(* IEC 61131-3 sources: RL_MAR/experiments/comparison/llm4plc/results/gpt-4o-mini_20260506_100619/20260506_103717, 4 files *)

(* ---- generated_code_iteration_0.st ---- *)
ructured-text
START_ST
FUNCTION_BLOCK SolarPanelTracking
VAR
    PanelAngle : REAL; (* Output for adjusting the solar panel angle *)
    SunriseTime : TIME := T#6H; (* Set the time for sunrise (6:00 AM) *)
    SunsetTime : TIME := T#18H; (* Set the time for sunset (6:00 PM) *)
    NoonTime : TIME := T#12H; (* Set the time for solar noon (12:00 PM) *)
    MorningAngle : REAL := 30.0; (* Set the morning angle for panels *)
    NoonAngle : REAL := 60.0; (* Set the noon angle for panels *)
    EveningAngle : REAL := 30.0; (* Set the evening angle for panels *)
    state : INT; (* The state variable *)
    prevState : INT; (* The previous state variable *)
END_VAR

VAR_INPUT
    CurrentTime : TIME; (* Input for current time *)
    SolarIntensity : REAL; (* Input for solar intensity *)
END_VAR

(* State Definitions *)
STATE_NIGHTTIME : INT := 0;
STATE_MORNING : INT := 1;
STATE_AFTERNOON_EVENING : INT := 2;
STATE_SOLAR_INTENSITY_OVERRIDE : INT := 3;

(* Main Logic *)
IF SolarIntensity >= 90.0 THEN
    PanelAngle := NoonAngle; (* Override to noon angle if solar intensity is high *)
    state := STATE_SOLAR_INTENSITY_OVERRIDE;
ELSE
    (* Determine the current state based on time *)
    IF CurrentTime < SunriseTime OR CurrentTime >= SunsetTime THEN
        PanelAngle := 0.0; (* Nighttime *)
        state := STATE_NIGHTTIME;
    ELSIF CurrentTime >= SunriseTime AND CurrentTime < NoonTime THEN
        PanelAngle := MorningAngle; (* Morning *)
        state := STATE_MORNING;
    ELSIF CurrentTime >= NoonTime AND CurrentTime < SunsetTime THEN
        PanelAngle := EveningAngle; (* Afternoon/Evening *)
        state := STATE_AFTERNOON_EVENING;
    END_IF;
END_IF;

(* State Transitions *)
CASE state OF
    STATE_NIGHTTIME:
        IF CurrentTime >= SunriseTime AND CurrentTime < NoonTime THEN
            state := STATE_MORNING; (* Transition to morning *)
        END_IF;
    STATE_MORNING:
        IF CurrentTime >= NoonTime AND CurrentTime < SunsetTime THEN
            state := STATE_AFTERNOON_EVENING; (* Transition to afternoon/evening *)
        END_IF;
    STATE_AFTERNOON_EVENING:
        IF CurrentTime >= SunsetTime THEN
            state := STATE_NIGHTTIME; (* Transition to nighttime *)
        END_IF;
END_CASE;

END_FUNCTION_BLOCK
END_ST

(* ---- generated_code_iteration_1.st ---- *)
START_REASON
The errors in the original Structured Text (ST) code occurred due to the incorrect use of the `VAR_INPUT` section. The variable declarations for input variables should be placed within the `VAR` section instead of `VAR_INPUT`. Additionally, the state definitions should be declared as constants or within the appropriate scope. The feedback indicated an unexpected token 'INT', which likely arose from the incorrect structure of the variable declarations. I will correct these issues while maintaining the function block structure.
END_REASON

START_ST
FUNCTION_BLOCK SolarPanelTracking
VAR
    PanelAngle : REAL; (* Output for adjusting the solar panel angle *)
    SunriseTime : TIME := T#6H; (* Set the time for sunrise (6:00 AM) *)
    SunsetTime : TIME := T#18H; (* Set the time for sunset (6:00 PM) *)
    NoonTime : TIME := T#12H; (* Set the time for solar noon (12:00 PM) *)
    MorningAngle : REAL := 30.0; (* Set the morning angle for panels *)
    NoonAngle : REAL := 60.0; (* Set the noon angle for panels *)
    EveningAngle : REAL := 30.0; (* Set the evening angle for panels *)
    state : INT; (* The state variable *)
    prevState : INT; (* The previous state variable *)
    CurrentTime : TIME; (* Input for current time *)
    SolarIntensity : REAL; (* Input for solar intensity *)
END_VAR

(* State Definitions *)
CONST
    STATE_NIGHTTIME : INT := 0;
    STATE_MORNING : INT := 1;
    STATE_AFTERNOON_EVENING : INT := 2;
    STATE_SOLAR_INTENSITY_OVERRIDE : INT := 3;
END_CONST

(* Main Logic *)
IF SolarIntensity >= 90.0 THEN
    PanelAngle := NoonAngle; (* Override to noon angle if solar intensity is high *)
    state := STATE_SOLAR_INTENSITY_OVERRIDE;
ELSE
    (* Determine the current state based on time *)
    IF CurrentTime < SunriseTime OR CurrentTime >= SunsetTime THEN
        PanelAngle := 0.0; (* Nighttime *)
        state := STATE_NIGHTTIME;
    ELSIF CurrentTime >= SunriseTime AND CurrentTime < NoonTime THEN
        PanelAngle := MorningAngle; (* Morning *)
        state := STATE_MORNING;
    ELSIF CurrentTime >= NoonTime AND CurrentTime < SunsetTime THEN
        PanelAngle := EveningAngle; (* Afternoon/Evening *)
        state := STATE_AFTERNOON_EVENING;
    END_IF;
END_IF;

(* State Transitions *)
CASE state OF
    STATE_NIGHTTIME:
        IF CurrentTime >= SunriseTime AND CurrentTime < NoonTime THEN
            state := STATE_MORNING; (* Transition to morning *)
        END_IF;
    STATE_MORNING:
        IF CurrentTime >= NoonTime AND CurrentTime < SunsetTime THEN
            state := STATE_AFTERNOON_EVENING; (* Transition to afternoon/evening *)
        END_IF;
    STATE_AFTERNOON_EVENING:
        IF CurrentTime >= SunsetTime THEN
            state := STATE_NIGHTTIME; (* Transition to nighttime *)
        END_IF;
END_CASE;

END_FUNCTION_BLOCK
END_ST

(* ---- generated_code_iteration_2.st ---- *)
START_REASON
The errors in the original Structured Text (ST) code occurred due to the incorrect use of the `VAR_INPUT` section. The variable declarations for input variables should be placed within the `VAR` section instead of `VAR_INPUT`. Additionally, the state definitions should be declared as constants or within the appropriate scope. The feedback indicated an unexpected token 'INT', which likely arose from the incorrect structure of the variable declarations. Furthermore, the feedback specified that a semicolon should replace 'STATE_NIGHTTIME', indicating a syntax issue in the CASE statement. I will correct these issues while maintaining the function block structure.
END_REASON

START_ST
FUNCTION_BLOCK SolarPanelTracking
VAR
    PanelAngle : REAL; (* Output for adjusting the solar panel angle *)
    SunriseTime : TIME := T#6H; (* Set the time for sunrise (6:00 AM) *)
    SunsetTime : TIME := T#18H; (* Set the time for sunset (6:00 PM) *)
    NoonTime : TIME := T#12H; (* Set the time for solar noon (12:00 PM) *)
    MorningAngle : REAL := 30.0; (* Set the morning angle for panels *)
    NoonAngle : REAL := 60.0; (* Set the noon angle for panels *)
    EveningAngle : REAL := 30.0; (* Set the evening angle for panels *)
    state : INT; (* The state variable *)
    prevState : INT; (* The previous state variable *)
    CurrentTime : TIME; (* Input for current time *)
    SolarIntensity : REAL; (* Input for solar intensity *)
END_VAR

(* State Definitions *)
CONST
    STATE_NIGHTTIME : INT := 0;
    STATE_MORNING : INT := 1;
    STATE_AFTERNOON_EVENING : INT := 2;
    STATE_SOLAR_INTENSITY_OVERRIDE : INT := 3;
END_CONST

(* Main Logic *)
IF SolarIntensity >= 90.0 THEN
    PanelAngle := NoonAngle; (* Override to noon angle if solar intensity is high *)
    state := STATE_SOLAR_INTENSITY_OVERRIDE;
ELSE
    (* Determine the current state based on time *)
    IF CurrentTime < SunriseTime OR CurrentTime >= SunsetTime THEN
        PanelAngle := 0.0; (* Nighttime *)
        state := STATE_NIGHTTIME;
    ELSIF CurrentTime >= SunriseTime AND CurrentTime < NoonTime THEN
        PanelAngle := MorningAngle; (* Morning *)
        state := STATE_MORNING;
    ELSIF CurrentTime >= NoonTime AND CurrentTime < SunsetTime THEN
        PanelAngle := EveningAngle; (* Afternoon/Evening *)
        state := STATE_AFTERNOON_EVENING;
    END_IF;
END_IF;

(* State Transitions *)
CASE state OF
    STATE_NIGHTTIME:
        IF CurrentTime >= SunriseTime AND CurrentTime < NoonTime THEN
            state := STATE_MORNING; (* Transition to morning *)
        END_IF;
    STATE_MORNING:
        IF CurrentTime >= NoonTime AND CurrentTime < SunsetTime THEN
            state := STATE_AFTERNOON_EVENING; (* Transition to afternoon/evening *)
        END_IF;
    STATE_AFTERNOON_EVENING:
        IF CurrentTime >= SunsetTime THEN
            state := STATE_NIGHTTIME; (* Transition to nighttime *)
        END_IF;
END_CASE;

END_FUNCTION_BLOCK
END_ST

(* ---- generated_code_iteration_3.st ---- *)
START_REASON
The errors in the original Structured Text (ST) code were primarily due to the incorrect syntax in the CASE statement where a semicolon was expected instead of the state name. This led to a compilation error in the CODESYS environment. Additionally, the structure of the variable declarations was correct, but I need to ensure that the CASE statement is properly formatted. I will correct the syntax issue in the CASE statement and ensure the overall structure adheres to the requirements.
END_REASON

START_ST
FUNCTION_BLOCK SolarPanelTracking
VAR
    PanelAngle : REAL; (* Output for adjusting the solar panel angle *)
    SunriseTime : TIME := T#6H; (* Set the time for sunrise (6:00 AM) *)
    SunsetTime : TIME := T#18H; (* Set the time for sunset (6:00 PM) *)
    NoonTime : TIME := T#12H; (* Set the time for solar noon (12:00 PM) *)
    MorningAngle : REAL := 30.0; (* Set the morning angle for panels *)
    NoonAngle : REAL := 60.0; (* Set the noon angle for panels *)
    EveningAngle : REAL := 30.0; (* Set the evening angle for panels *)
    state : INT; (* The state variable *)
    prevState : INT; (* The previous state variable *)
    CurrentTime : TIME; (* Input for current time *)
    SolarIntensity : REAL; (* Input for solar intensity *)
END_VAR

(* State Definitions *)
CONST
    STATE_NIGHTTIME : INT := 0;
    STATE_MORNING : INT := 1;
    STATE_AFTERNOON_EVENING : INT := 2;
    STATE_SOLAR_INTENSITY_OVERRIDE : INT := 3;
END_CONST

(* Main Logic *)
IF SolarIntensity >= 90.0 THEN
    PanelAngle := NoonAngle; (* Override to noon angle if solar intensity is high *)
    state := STATE_SOLAR_INTENSITY_OVERRIDE;
ELSE
    (* Determine the current state based on time *)
    IF CurrentTime < SunriseTime OR CurrentTime >= SunsetTime THEN
        PanelAngle := 0.0; (* Nighttime *)
        state := STATE_NIGHTTIME;
    ELSIF CurrentTime >= SunriseTime AND CurrentTime < NoonTime THEN
        PanelAngle := MorningAngle; (* Morning *)
        state := STATE_MORNING;
    ELSIF CurrentTime >= NoonTime AND CurrentTime < SunsetTime THEN
        PanelAngle := EveningAngle; (* Afternoon/Evening *)
        state := STATE_AFTERNOON_EVENING;
    END_IF;
END_IF;

(* State Transitions *)
CASE state OF
    STATE_NIGHTTIME:
        IF CurrentTime >= SunriseTime AND CurrentTime < NoonTime THEN
            state := STATE_MORNING; (* Transition to morning *)
        END_IF;
    STATE_MORNING:
        IF CurrentTime >= NoonTime AND CurrentTime < SunsetTime THEN
            state := STATE_AFTERNOON_EVENING; (* Transition to afternoon/evening *)
        END_IF;
    STATE_AFTERNOON_EVENING:
        IF CurrentTime >= SunsetTime THEN
            state := STATE_NIGHTTIME; (* Transition to nighttime *)
        END_IF;
    STATE_SOLAR_INTENSITY_OVERRIDE: (* Added missing case for solar intensity override *)
        IF SolarIntensity < 90.0 THEN
            state := STATE_NIGHTTIME; (* Transition back to nighttime if intensity drops *)
        END_IF;
END_CASE;

END_FUNCTION_BLOCK
END_ST
